Staubli VAL3: cartStatus.pgx

public program cartStatus(num x_nCartConnFlag, num x_nLastMsgAge)
begin

  // update connection status on port 11001 (cartesian server)

  gotoxy(scMonitor, 0,1)
  put(scMonitor, "Port 11001:")
  gotoxy(scMonitor, 12,1)
  switch x_nCartConnFlag
    case -1
      put(scMonitor, "connection lost")
    break
    case 0
      put(scMonitor, "not connected")
    break
    case 1
      put(scMonitor, "connected")
    break
    default
      put(scMonitor, "not connected")
    break
  endSwitch

  gotoxy(scMonitor, 0,2)
  put(scMonitor, "Last cart msg:")
  gotoxy(scMonitor, 14,2)
  if (x_nLastMsgAge < 0)
    put(scMonitor, "n/a")
  else
    put(scMonitor, toString(".1", x_nLastMsgAge) + " s")
  endIf

end
